Yaskawa INFORM job: R1_S1_SEC.JBI

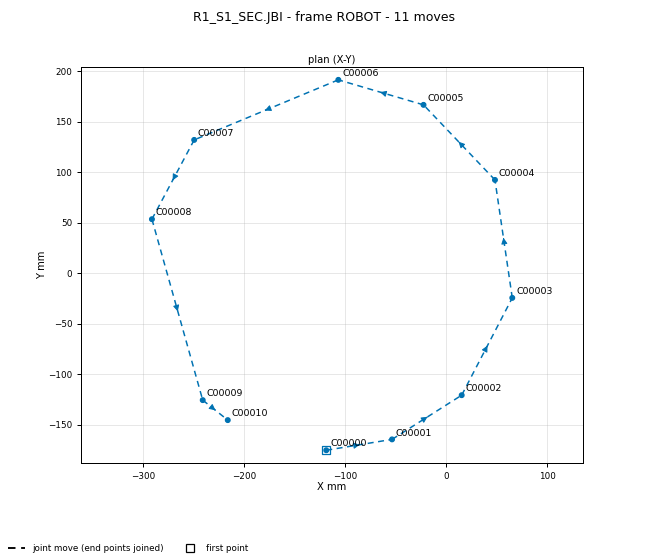
[picture p0: tool path of R1_S1_SEC.JBI in frame ROBOT, 11 of 11 moves have a stored position in this frame; points joined in program order, loops and branches not executed]
/JOB
//NAME R1_S1_SEC
///FOLDERNAME INNE
//POS
///NPOS 11,11,0,0,0,0
///TOOL 0
///POSTYPE ROBOT
///RECTAN
///RCONF 0,0,0,0,0,0,0,0,0,0,0,0,0,0,0,0,0,0,0,0,0,0,0,0
C00000=-118.710,-175.290,-2196.473,-0.0001,-0.0023,179.9973
C00001=-53.541,-164.519,-2196.335,-0.0147,0.0049,-179.9922
C00002=15.485,-120.735,-2197.065,-0.0170,0.0014,-179.9907
C00003=65.588,-24.325,-2197.250,-0.0156,0.0007,-179.9880
C00004=48.435,92.550,-2197.439,-0.0149,0.0006,-179.9891
C00005=-22.351,166.930,-2197.403,-0.0137,-0.0019,-179.9953
C00006=-106.762,191.707,-2197.202,-0.0129,-0.0047,179.9941
C00007=-249.579,132.208,-2196.926,-0.0132,-0.0051,179.9957
C00008=-291.443,53.644,-2197.036,-0.0140,-0.0051,179.9994
C00009=-241.115,-125.625,-2196.017,-0.0199,-0.0049,179.9987
C00010=-216.300,-145.437,-2195.953,-0.0172,-0.0044,179.9984
BC00000=1472.925,829.369,1292.692
BC00001=1472.925,829.369,1292.692
BC00002=1472.925,829.369,1292.692
BC00003=1472.925,829.369,1292.692
BC00004=1472.925,829.369,1292.692
BC00005=1472.925,829.369,1292.692
BC00006=1472.925,829.369,1292.692
BC00007=1472.925,829.369,1292.692
BC00008=1472.925,829.369,1292.692
BC00009=1472.925,829.369,1292.692
BC00010=1472.925,829.369,1292.692
//INST
///DATE 2023/10/04 15:16
///ATTR SC,RW,RJ
////FRAME ROBOT
///GROUP1 RB1,BS1
NOP
MOVJ C00000 BC00000 VJ=0.78
MOVJ C00001 BC00001 VJ=0.78
MOVJ C00002 BC00002 VJ=0.78
MOVJ C00003 BC00003 VJ=0.78
MOVJ C00004 BC00004 VJ=0.78
MOVJ C00005 BC00005 VJ=0.78
MOVJ C00006 BC00006 VJ=0.78
MOVJ C00007 BC00007 VJ=0.78
MOVJ C00008 BC00008 VJ=0.78
MOVJ C00009 BC00009 VJ=0.78
MOVJ C00010 BC00010 VJ=0.78
END
